// TwinCAT 3 PLC project PLC
// ProgramVersion: 3.1.4024.0
// libraries:
//   Tc2_Standard, * (Beckhoff Automation GmbH)
//   Tc2_System, * (Beckhoff Automation GmbH)
//   Tc3_Module, * (Beckhoff Automation GmbH)
// project tree:
//   / GlobalTextList.TcGTLO, PlcTask.TcTTO, Visualization Manager.TcVMO (not stored), Visualization.TcVIS
//   GVLs/ GVL.TcGVL
//   POUs/ MAIN_SFC.TcPOU
// real-time tasks:
//   TASK PlcTask: cycle T#10ms, priority 20, ADS port 350

CONFIGURATION PLC
    RESOURCE PLC ON TwinCAT3
        TASK PlcTask(INTERVAL := T#10ms, PRIORITY := 20);
        PROGRAM MAIN_SFC WITH PlcTask : MAIN_SFC;
    END_RESOURCE
END_CONFIGURATION

// ---- GVLs/GVL.TcGVL
{attribute 'qualified_only'}
VAR_GLOBAL
	StartButton			: BOOL;
	CarRedLight			: BOOL;
	CarYellowLight		: BOOL;
	CarGreenLight		: BOOL;
	CrossWalkRedLight	: BOOL;
	CrossWalkGreenLight : BOOL;
	NightLight			: BOOL; 
END_VAR

// ---- POUs/MAIN_SFC.TcPOU
PROGRAM MAIN_SFC
VAR

END_VAR

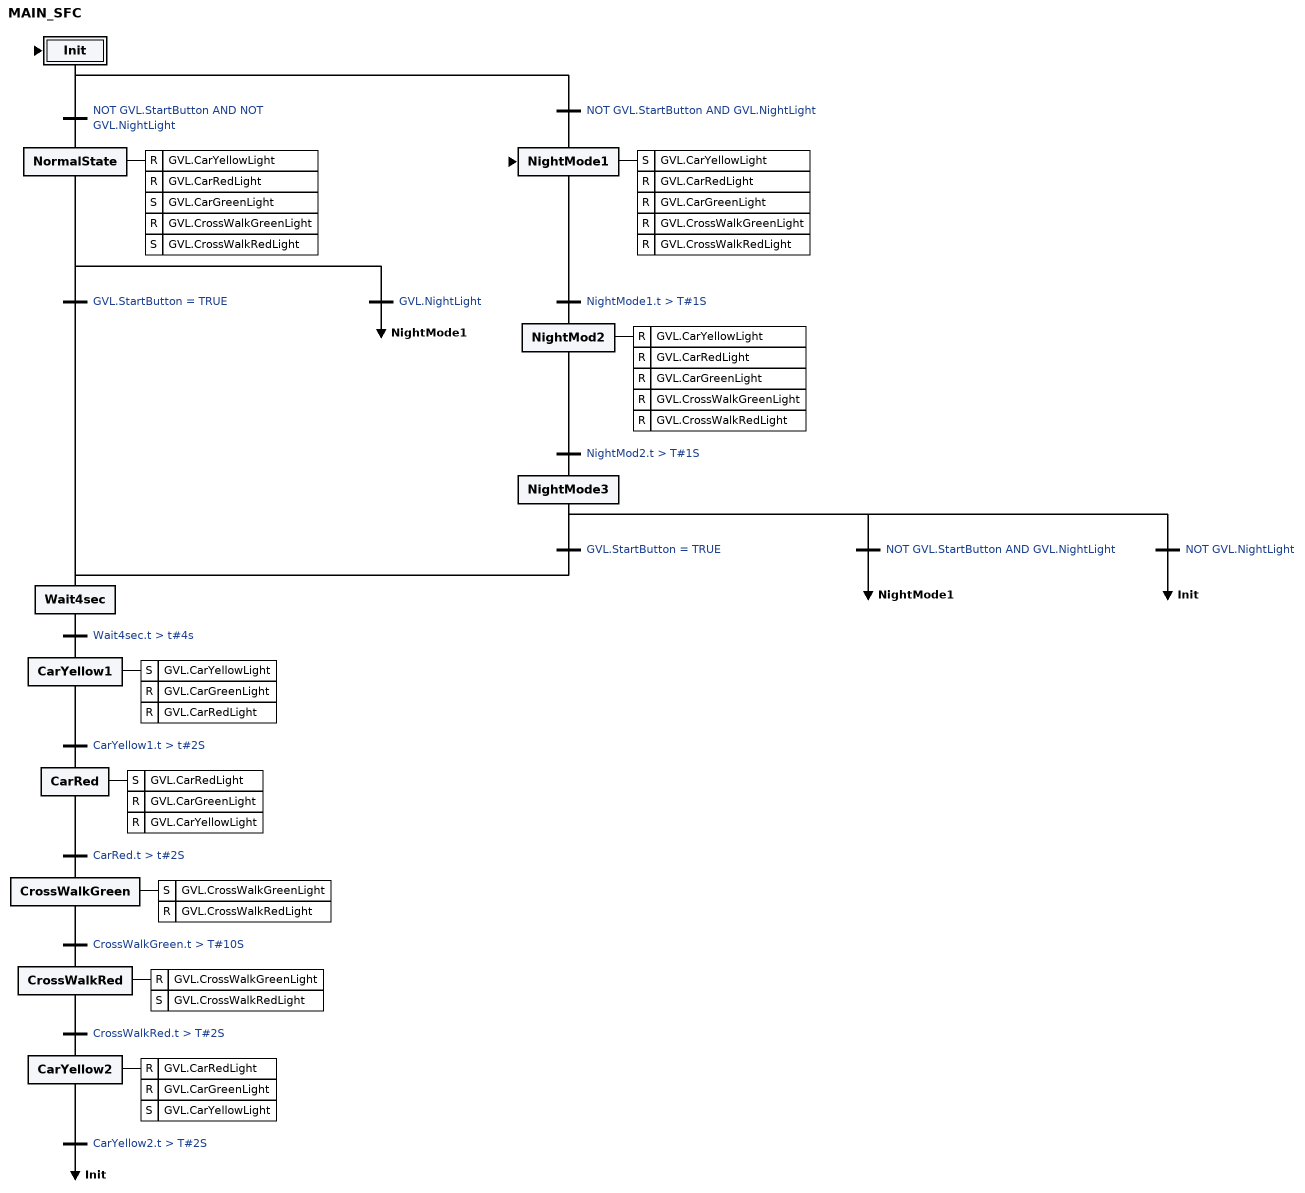
INITIAL_STEP Init:
END_STEP
TRANSITION FROM Init TO NormalState
    := NOT GVL.StartButton AND NOT GVL.NightLight;
END_TRANSITION
STEP NormalState:
    GVL.CarYellowLight(R);
    GVL.CarRedLight(R);
    GVL.CarGreenLight(S);
    GVL.CrossWalkGreenLight(R);
    GVL.CrossWalkRedLight(S);
END_STEP
TRANSITION FROM NormalState TO Wait4sec
    := GVL.StartButton = TRUE;
END_TRANSITION
TRANSITION FROM NormalState TO NightMode1
    := GVL.NightLight;
END_TRANSITION
TRANSITION FROM Init TO NightMode1
    := NOT GVL.StartButton AND GVL.NightLight;
END_TRANSITION
STEP NightMode1:
    GVL.CarYellowLight(S);
    GVL.CarRedLight(R);
    GVL.CarGreenLight(R);
    GVL.CrossWalkGreenLight(R);
    GVL.CrossWalkRedLight(R);
END_STEP
TRANSITION FROM NightMode1 TO NightMod2
    := NightMode1.t > T#1S;
END_TRANSITION
STEP NightMod2:
    GVL.CarYellowLight(R);
    GVL.CarRedLight(R);
    GVL.CarGreenLight(R);
    GVL.CrossWalkGreenLight(R);
    GVL.CrossWalkRedLight(R);
END_STEP
TRANSITION FROM NightMod2 TO NightMode3
    := NightMod2.t > T#1S;
END_TRANSITION
STEP NightMode3:
END_STEP
TRANSITION FROM NightMode3 TO Wait4sec
    := GVL.StartButton = TRUE;
END_TRANSITION
TRANSITION FROM NightMode3 TO NightMode1
    := NOT GVL.StartButton AND GVL.NightLight;
END_TRANSITION
TRANSITION FROM NightMode3 TO Init
    := NOT GVL.NightLight;
END_TRANSITION
STEP Wait4sec:
END_STEP
TRANSITION FROM Wait4sec TO CarYellow1
    := Wait4sec.t > t#4s;
END_TRANSITION
STEP CarYellow1:
    GVL.CarYellowLight(S);
    GVL.CarGreenLight(R);
    GVL.CarRedLight(R);
END_STEP
TRANSITION FROM CarYellow1 TO CarRed
    := CarYellow1.t > t#2S;
END_TRANSITION
STEP CarRed:
    GVL.CarRedLight(S);
    GVL.CarGreenLight(R);
    GVL.CarYellowLight(R);
END_STEP
TRANSITION FROM CarRed TO CrossWalkGreen
    := CarRed.t > t#2S;
END_TRANSITION
STEP CrossWalkGreen:
    GVL.CrossWalkGreenLight(S);
    GVL.CrossWalkRedLight(R);
END_STEP
TRANSITION FROM CrossWalkGreen TO CrossWalkRed
    := CrossWalkGreen.t > T#10S;
END_TRANSITION
STEP CrossWalkRed:
    GVL.CrossWalkGreenLight(R);
    GVL.CrossWalkRedLight(S);
END_STEP
TRANSITION FROM CrossWalkRed TO CarYellow2
    := CrossWalkRed.t > T#2S;
END_TRANSITION
STEP CarYellow2:
    GVL.CarRedLight(R);
    GVL.CarGreenLight(R);
    GVL.CarYellowLight(S);
END_STEP
TRANSITION FROM CarYellow2 TO Init
    := CarYellow2.t > T#2S;
END_TRANSITION

END_PROGRAM

// ---- GlobalTextList.TcGTLO
TEXTLIST GlobalTextList
  609 = 'Night Light'
END_TEXTLIST

// ---- Visualization.TcVIS
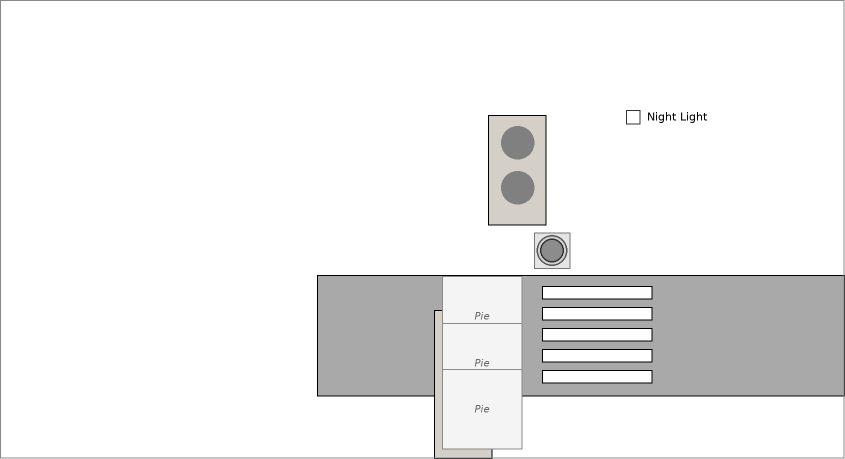
VISUALIZATION Visualization  // 845x459
    PushSwitch (534,232 36x37), variable: GVL.StartButton, behaviour: TAP, style: Switch-PushSwitch-Gray
    Rectangle (317,275 528x121)
    Checkbox (624,102 111x30), "Night Light", variable: GVL.NightLight
    Rectangle (542,286 110x13)
    Rectangle (542,307 110x13)
    Rectangle (542,328 110x13)
    Rectangle (542,349 110x13)
    Rectangle (542,370 110x13)
    Rectangle (488,115 58x110)
    Ellipse (500,125 35x35), colour toggle: GVL.CrossWalkRedLight
    Ellipse (500,170 35x35), colour toggle: GVL.CrossWalkGreenLight
    Rectangle (434,310 58x149)
    Pie (442,276 80x80), colour toggle: GVL.CarRedLight
    Pie (442,323 80x80), colour toggle: GVL.CarYellowLight
    Pie (442,369 80x80), colour toggle: GVL.CarGreenLight
END_VISUALIZATION
